// TIA Portal V19 export
TYPE "C501_VAR_IF_BBI_TYPIC"
   STRUCT
      REQ_UIT { ExternalAccessible := 'False'; ExternalVisible := 'False'; ExternalWritable := 'False'} : Bool;   // Aanvraag om regime Uit te activeren
      REQ_BWK { ExternalAccessible := 'False'; ExternalVisible := 'False'; ExternalWritable := 'False'} : Bool;   // Aanvraag om regime Bewaken te activeren
      REQ_BLUS1 { ExternalAccessible := 'False'; ExternalVisible := 'False'; ExternalWritable := 'False'} : Bool;   // Aanvraag om regime Blussen Hydrant te activeren
      REQ_BLUS2 { ExternalAccessible := 'False'; ExternalVisible := 'False'; ExternalWritable := 'False'} : Bool;   // Aanvraag om regime Blussen Hydrant en WMS te activeren
      REQ_TEST { ExternalAccessible := 'False'; ExternalVisible := 'False'; ExternalWritable := 'False'} : Bool;   // Aanvraag om regime Testen te activeren
      EXT_HW { ExternalAccessible := 'False'; ExternalVisible := 'False'; ExternalWritable := 'False'} : Bool;   // Sturings hardware (PLC) in storing
      STO { ExternalAccessible := 'False'; ExternalVisible := 'False'; ExternalWritable := 'False'} : Struct   // Opsomming van alle storingen
         A001 : Bool;   // Beveiliging aangesproken
         A002 : Bool;   // Beveiliging No-Break aangesproken
         A003 : Bool;   // Schuif ALSB uitgeschakeld
         A004 : Bool;   // Schuif ALSB in test
         A005 : Bool;   // Schuif ALSB uitgereden
         A006 : Bool;   // Lekdetectie in pomplokaal
         A007 : Bool;   // Overspanningsbeveiliging aangesproken
         A008 : Bool;   // Beveiliging kastklimatisatie aangesproken
         A009 : Bool;   // Lastscheider niet aan
      END_STRUCT;
   END_STRUCT;
END_TYPE
